KUKA KRL program: Mes_Loop_Main.src

&ACCESS RVP
&REL 2
DEF Mes_Loop_Main( )

Mes_InFo_Int()
loop
Mes_InFo_Main()

WAIT SEC 0
endloop


END
